// TwinCAT 3 PLC project gearln
// ProgramVersion: 3.1.4024.0
// libraries:
//   Tc2_MC2, * (Beckhoff Automation GmbH)
//   Tc2_Standard, * (Beckhoff Automation GmbH)
//   Tc2_System, * (Beckhoff Automation GmbH)
//   Tc3_Module, * (Beckhoff Automation GmbH)
// project tree:
//   / PlcTask.TcTTO
//   POUs/ MAIN.TcPOU
// real-time tasks:
//   TASK PlcTask: cycle T#10ms, priority 20, ADS port 350
// motion (NC):
//   TASK NC-Task 1 SAF: cycle T#2ms, priority 4, ADS port 501
//   TASK NC-Task 1 SVB: cycle T#10ms, priority 8, ADS port 511
//   AXIS Axis 1 (id 1)
//     OtherSettings: AllowMotionCmdToSlave=true
//     encoder EncType=1
//     drive DrvType=5
//       Analog: TorqueSetpointScale=10, ScaleFactorActTorque=0.1
//       TimeComp: TaskDelayCycles=1
//     controller CtrType=1
//       CtrPara: PriorControlFactor=1
//         Observer: BandWidth=20
//   AXIS Axis 2 (id 2)
//     OtherSettings: AllowMotionCmdToSlave=true
//     encoder EncType=1
//     drive DrvType=5
//       Analog: TorqueSetpointScale=10, ScaleFactorActTorque=0.1
//       TimeComp: TaskDelayCycles=1
//     controller CtrType=1
//       CtrPara: PriorControlFactor=1
//         Observer: BandWidth=20
// variable links:
//   gearln/gearln Instance <-> NC-Task 1 SAF/Axes/Axis 1
//     PlcTask Inputs/MAIN.master.NcToPlc <-> Outputs/ToPlc
//     PlcTask Outputs/MAIN.master.PlcToNc <-> Inputs/FromPlc
//   gearln/gearln Instance <-> NC-Task 1 SAF/Axes/Axis 2
//     PlcTask Inputs/MAIN.slave.NcToPlc <-> Outputs/ToPlc
//     PlcTask Outputs/MAIN.slave.PlcToNc <-> Inputs/FromPlc

CONFIGURATION gearln
    RESOURCE PLC ON TwinCAT3
        TASK PlcTask(INTERVAL := T#10ms, PRIORITY := 20);
        PROGRAM MAIN WITH PlcTask : MAIN;
    END_RESOURCE
END_CONFIGURATION

// ---- POUs/MAIN.TcPOU
PROGRAM MAIN
VAR
	master 		: AXIS_REF;
	slave 		: AXIS_REF;
	fb_Power	: MC_Power;
	bEnable		: BOOL;
	fb_Power2	: MC_Power;
	fb_GearIn	: MC_GearIn;
	enable		: BOOL;
	fbMove 		: MC_MoveAbsolute;
	mEnable		: BOOL;
	fb_GearOut	: MC_GearOut;
	nenable		: BOOL;
	fb_Stop		: MC_Stop;
	fb_halt 	:MC_Halt;
	bStop 		: BOOL:=FALSE;
	deger 		: LREAL;

	d: BOOL;
	dEnable: BOOL;
END_VAR


fb_Power(//For master
	Axis:=master , 
	Enable:= bEnable, 
	Enable_Positive:= bEnable, 
	Enable_Negative:= bEnable, 
	Override:=100 );
	
fb_Power2(//for slave
	Axis:=slave , 
	Enable:=bEnable , 
	Enable_Positive:=bEnable , 
	Enable_Negative:= bEnable, 
	Override:=100 );
	

fb_GearIn(
	Master:=master , 
	Slave:= slave, 
	Execute:= enable, 
	RatioNumerator:=5 , 
	RatioDenominator:= 1);
	
fbMove(
	Axis:=master , 
	Execute:=mEnable , 
	Position:=deger , 
	Velocity:= 100 );
	
	
fb_GearOut(
	Slave:= slave, 
	Execute:=nenable);
	
fb_Stop(
	Axis:= master, 
	Execute:=bStop);
	

fb_halt(
	Axis:=master , 
	Execute:= dEnable);

END_PROGRAM
